PROGRAM p_slow_task
VAR
END_VAR

(*Programmaufrufte im slow Task (10ms)*)
//Call Slow Tasks for Lynus 	
MqttCommunicator();
p_Datenschnittstelle_L();


//Stefan Lackner 14.02.2023
PrgModbus();		// Modbus TCP functions
PrgEMS();			// EMS Fucntion

END_PROGRAM

(* stored: Version 1.1.0.1, ProductVersion 3.1.4024.3
   POU p_slow_task: Id {71817dfd-8862-47d0-b3a3-29d0dd89b5fb}, SpecialFunc None *)
